Fanuc KAREL source: kx00012.KL

-- PROVISIONAL review KL for V940-1; original PC SHA256 b5fca54fbf779efeab8b306f9ee620bbcdc1c7c53e21f5c99aeb104323a47af3
-- Incomplete behavior may be omitted. Consult companion uncertainty JSON. Do not deploy.
PROGRAM KX00012
%NOLOCKGROUP
VAR
  I : INTEGER
  J : INTEGER
  B : BOOLEAN
  F : FILE
  S : STRING[80]
-- UNRESOLVED_DECL P type=000102
BEGIN
  -- V9_ZERO_TABLE_METADATA_HINT layout=0001; no indexed target words; source/name/runtime held
  -- UNRESOLVED_PC offsets 5-7; opcodes 9C,66
  -- UNRESOLVED_PC offsets 12-16; opcodes 7F
END KX00012
